// TIA Portal V20 export
FUNCTION_BLOCK "FB_LoaderFixture"   // FB207, SCL
{ S7_Optimized_Access := 'TRUE' }
// stored: AutoNumber false, MemoryReserve 100, SetENOAutomatically false
   VAR_INPUT
      iAxisV_Moving : Bool;
      iAxisV_InPos : Bool;
      iAxisW_Moving : Bool;
      iAxisW_InPos : Bool;
   END_VAR
   VAR_OUTPUT
      oFixtureOpenReq : Bool;
      oFixtureCloseReq : Bool;
      oLoadGripperOpenReq : Bool;
      oUnloadGripperCloseReq : Bool;
      oBlowingReq : Bool;
      oAxisV_StartReq : Bool;
      oAxisV_PosSetPoint : Real;
      oAxisW_StartReq : Bool;
      oAxisW_PosSetPoint : Real;
   END_VAR
   VAR
      sFixtureMain : "FB_FixtureUnloadLoad";
      sFixtureUnloading { S7_SetPoint := 'True'} : "FB_FixtureUnloading";
      sFixtureLoading { S7_SetPoint := 'True'} : "FB_FixtureLoading";
      sFixtureBlowing { S7_SetPoint := 'True'} : "FB_FixtureBlowing";
      sFixtureRelease { S7_SetPoint := 'True'} : "FB_FixtureRelease";
      sFixtureV_Init { S7_SetPoint := 'True'} : "FB_FixtureV_Init";
      sFixtureW_Init { S7_SetPoint := 'True'} : "FB_FixtureW_Init";
      sAxisVSafePos { S7_SetPoint := 'True'} : LReal;
      sStepPauseSeq { S7_SetPoint := 'True'} : Bool;
   END_VAR
   VAR_TEMP
      tAxisV_Position : Struct
         FixtureLoad : Bool;
         FixtureUnload : Bool;
         FixtureBlowing : Bool;
         FixtureSafe : Bool;
         ShuttleSafe : Bool;
         Shuttle1Blowing : Bool;
      END_STRUCT;
      tAxisW_Position : Struct
         FixtureLoad : Bool;
         FixtureUnload : Bool;
         FixtureBlowing : Bool;
         FixtureSafe : Bool;
         Approach : Bool;
      END_STRUCT;
   END_VAR
BEGIN
   REGION Axis V Safe Position
       IF "DB_LoaderShuttle1".sShuttlePosInt THEN
           #sAxisVSafePos := "DB_AxisPosMachinePLC".Axis_V.Shuttle_1.LoadUnload;
       ELSIF "DB_LoaderShuttle2".sShuttlePosInt THEN
           #sAxisVSafePos := "DB_AxisPosMachinePLC".Axis_V.Shuttle_2.LoadUnload;
       ELSE
           #sAxisVSafePos := "DB_AxisPosMachinePLC".Axis_V.Fixture.Safe;
       END_IF;
       // WFA revoir la gestion du Setpoint Safe en foncton de la shuttle
       #sAxisVSafePos := "DB_AxisPosMachinePLC".Axis_V.Fixture.Safe;
   END_REGION

   REGION Position Check
       REGION Axis V
           // Position : Fixture Load
           "FC_PositionCheck"(iAxisCurrentPos := "DB_AxisPosition".sAxis07_V."$AA_IM",
                              iAxisTargetPos := "DB_AxisPosMachinePLC".Axis_V.Fixture.Load,
                              iTolMin := 0.001,
                              iTolMax := 0.001,
                              iInPos => #tAxisV_Position.FixtureLoad);

           // Position : Fixture Unload
           "FC_PositionCheck"(iAxisCurrentPos := "DB_AxisPosition".sAxis07_V."$AA_IM",
                              iAxisTargetPos := "DB_AxisPosMachinePLC".Axis_V.Fixture.Unload,
                              iTolMin := 0.001,
                              iTolMax := 0.001,
                              iInPos => #tAxisV_Position.FixtureUnload);

           // Position : Fixture Blowing
           "FC_PositionCheck"(iAxisCurrentPos := "DB_AxisPosition".sAxis07_V."$AA_IM",
                              iAxisTargetPos := "DB_AxisPosMachinePLC".Axis_V.Fixture.Blowing,
                              iTolMin := 0.001,
                              iTolMax := 0.001,
                              iInPos => #tAxisV_Position.FixtureBlowing);

           // Position : Fixture Safe
           "FC_PositionCheck"(iAxisCurrentPos := "DB_AxisPosition".sAxis07_V."$AA_IM",
                              iAxisTargetPos := #sAxisVSafePos,
                              iTolMin := 0.001,
                              iTolMax := 0.001,
                              iInPos => #tAxisV_Position.FixtureSafe);

           // Position : Safe (Shuttle)
           "FC_PositionCheck"(iAxisCurrentPos := "DB_AxisPosition".sAxis07_V."$AA_IM",
                              iAxisTargetPos := "DB_AxisPosMachinePLC".Axis_V.Safe,
                              iTolMin := 0.001,
                              iTolMax := 0.001,
                              iInPos => #tAxisV_Position.ShuttleSafe);

           // Position : Blowing Shuttle 1
           "FC_PositionCheck"(iAxisCurrentPos := "DB_AxisPosition".sAxis07_V."$AA_IM",
                              iAxisTargetPos := "DB_AxisPosMachinePLC".Axis_V.Shuttle_1.Blowing,
                              iTolMin := 0.001,
                              iTolMax := 0.001,
                              iInPos => #tAxisV_Position.Shuttle1Blowing);
       END_REGION

       REGION Axis W
           // Position : Fixture Load
           "FC_PositionCheck"(iAxisCurrentPos := "DB_AxisPosition".sAxis08_W."$AA_IM",
                              iAxisTargetPos := "DB_AxisPosMachinePLC".Axis_W.Fixture.Load,
                              iTolMin := 0.001,
                              iTolMax := 0.001,
                              iInPos => #tAxisW_Position.FixtureLoad);

           // Position : Fixture Unload
           "FC_PositionCheck"(iAxisCurrentPos := "DB_AxisPosition".sAxis08_W."$AA_IM",
                              iAxisTargetPos := "DB_AxisPosMachinePLC".Axis_W.Fixture.Unload,
                              iTolMin := 0.001,
                              iTolMax := 0.001,
                              iInPos => #tAxisW_Position.FixtureUnload);

           // Position : Fixture Blowing
           "FC_PositionCheck"(iAxisCurrentPos := "DB_AxisPosition".sAxis08_W."$AA_IM",
                              iAxisTargetPos := "DB_AxisPosMachinePLC".Axis_W.Fixture.Blowing,
                              iTolMin := 0.001,
                              iTolMax := 0.001,
                              iInPos => #tAxisW_Position.FixtureBlowing);

           // Position : Fixture Safe
           "FC_PositionCheck"(iAxisCurrentPos := "DB_AxisPosition".sAxis08_W."$AA_IM",
                              iAxisTargetPos := "DB_AxisPosMachinePLC".Axis_W.Fixture.Safe,
                              iTolMin := 0.001,
                              iTolMax := 0.001,
                              iInPos => #tAxisW_Position.FixtureSafe);

           // Position : Approach (confondu avec load/unload)
           "FC_PositionCheck"(iAxisCurrentPos := "DB_AxisPosition".sAxis08_W."$AA_IM",
                              iAxisTargetPos := "DB_AxisPosMachinePLC".Axis_W.Fixture.Approach,
                              iTolMin := 0.001,
                              iTolMax := 0.001,
                              iInPos => #tAxisW_Position.Approach);
       END_REGION
   END_REGION

   REGION Step Pause Sequence
       #sStepPauseSeq := "LBP_ModeGroup".E_JOG OR "DB_ExtraMissingPart".sGlobalExtraMissing;

       #sFixtureUnloading.iStepPause := #sStepPauseSeq;
       #sFixtureLoading.iStepPause := #sStepPauseSeq;
       #sFixtureBlowing.iStepPause := #sStepPauseSeq;
       #sFixtureRelease.iStepPause := #sStepPauseSeq;
       #sFixtureV_Init.iStepPause := #sStepPauseSeq;
       #sFixtureW_Init.iStepPause := #sStepPauseSeq;
   END_REGION

   REGION Fixture Unload Load
       // M33 : Fixture Unloading Request
       #sFixtureMain.iFixtureUnloadingRequest := "LBP_Chan1".MDyn[33];

       // M35 : Fixture Blowing Request
       #sFixtureMain.iFixtureBlowingRequest := "LBP_Chan1".MDyn[35];

       // M34 : Fixture Loading Request
       #sFixtureMain.iFixtureLoadingRequest := "LBP_Chan1".MDyn[34];

       // Release request (Release not used)
       #sFixtureMain.iFixtureReleaseRequest := FALSE;

       // M31 : Fixture V Init Request
       #sFixtureMain.iFixtureV_InitRequest := "LBP_Chan1".MDyn[31];

       // M32 : Fixture W Init Request
       #sFixtureMain.iFixtureW_InitRequest := "LBP_Chan1".MDyn[32];

       // Gripper ready for unloading
       #sFixtureMain.iGripperReadyForUnloading := ("DB_GestionGripper".sGripperStatus.Available OR "DB_GestionGripper".sGripperStatus.DrivedByFixture)
       AND ((NOT "DB_PartManagement".sPosition.sGripper.Drilled.Presence.Part AND NOT "DB_PartManagement".sPosition.sGripper.Drilled.Presence.BW AND "DB_GestionGripper".sDrilledGripper.oStateOpen AND "DB_WorkingModes".sEmptying)
       OR (NOT "DB_PartManagement".sPosition.sGripper.Drilled.Presence.Part AND NOT "DB_PartManagement".sPosition.sGripper.Drilled.Presence.BW AND "DB_PartManagement".sPosition.sGripper.Undrilled.Presence.Part AND "DB_PartManagement".sPosition.sGripper.Undrilled.Presence.BW AND "DB_GestionGripper".sDrilledGripper.oStateOpen AND "DB_WorkingModes".sNormal));

       // Gripper ready for loading
       #sFixtureMain.iGripperReadyForLoading := ("DB_GestionGripper".sGripperStatus.Available OR "DB_GestionGripper".sGripperStatus.DrivedByFixture)
       AND (("DB_PartManagement".sPosition.sGripper.Undrilled.Presence.Part AND "DB_PartManagement".sPosition.sGripper.Undrilled.Presence.BW AND "DB_WorkingModes".sFilling)
       OR ("DB_PartManagement".sPosition.sGripper.Undrilled.Presence.Part AND "DB_PartManagement".sPosition.sGripper.Undrilled.Presence.BW  AND ("DB_WorkingModes".sNormal OR "DB_WorkingModes".sEmptying)));

       // Gripper ready for blowing
       #sFixtureMain.iGripperReadyForBlowing := ("DB_GestionGripper".sGripperStatus.Available OR "DB_GestionGripper".sGripperStatus.DrivedByFixture)
       AND #sFixtureMain.iGripperReadyForLoading;

       // Gripper ready for Release (Release not used)
       #sFixtureMain.iGripperReadyForRelease := ("DB_GestionGripper".sGripperStatus.Available OR "DB_GestionGripper".sGripperStatus.DrivedByFixture);

       // Gripper ready for V Init
       #sFixtureMain.iGripperReadyForV_Init := ("DB_GestionGripper".sGripperStatus.Available OR "DB_GestionGripper".sGripperStatus.DrivedByFixture);

       // Gripper ready for W Init
       #sFixtureMain.iGripperReadyForW_Init := ("DB_GestionGripper".sGripperStatus.Available OR "DB_GestionGripper".sGripperStatus.DrivedByFixture);


       // Fixture ready for unloading
       #sFixtureMain.iFixtureReadyForUnloading := TRUE;

       // Fixture ready for loading
       #sFixtureMain.iFixtureReadyForLoading := "DB_PartManagement".sPosition.sFixtureEmpty;

       // Fixture ready for blowing
       #sFixtureMain.iFixtureReadyForBlowing := TRUE;

       // Fixture ready for Release (Release not used)
       #sFixtureMain.iFixtureReadyForRelease := TRUE;

       // Fixture ready for V Init
       #sFixtureMain.iFixtureReadyForV_Init := TRUE;

       // Fixture ready for W Init
       #sFixtureMain.iFixtureReadyForW_Init := TRUE;


       // Axis ready for Unloading
       #sFixtureMain.iAxisReadyForUnloading :=
       ("DB_AxisPosition".sAxis01_X."$AA_IM" = "DB_AxisPosMachineNC".Axis_X.Unload
       AND "DB_AxisPosition".sAxis02_Y."$AA_IM" = "DB_AxisPosMachineNC".Axis_Y.Unload
       AND "DB_AxisPosition".sAxis04_B."$AA_IM" = "DB_AxisPosMachineNC".Axis_B.Unload
       AND "DB_AxisPosition".sAxis03_ZM."$AA_IM" = "DB_AxisPosition".sAxis03_ZM."$MA_POS_LIMIT_MINUS2" + 1);

       // Axis ready for Loading
       #sFixtureMain.iAxisReadyForLoading :=
       ("DB_AxisPosition".sAxis01_X."$AA_IM" = "DB_AxisPosMachineNC".Axis_X.Load
       AND "DB_AxisPosition".sAxis02_Y."$AA_IM" = "DB_AxisPosMachineNC".Axis_Y.Load
       AND "DB_AxisPosition".sAxis04_B."$AA_IM" = "DB_AxisPosMachineNC".Axis_B.Load
       AND "DB_AxisPosition".sAxis03_ZM."$AA_IM" = "DB_AxisPosition".sAxis03_ZM."$MA_POS_LIMIT_MINUS2" + 1);

       // Axis ready for Blowing
       #sFixtureMain.iAxisReadyForBlowing :=
       ("DB_AxisPosition".sAxis01_X."$AA_IM" = "DB_AxisPosMachineNC".Axis_X.Blowing
       AND "DB_AxisPosition".sAxis02_Y."$AA_IM" = "DB_AxisPosMachineNC".Axis_Y.Blowing
       AND "DB_AxisPosition".sAxis04_B."$AA_IM" = "DB_AxisPosMachineNC".Axis_B.Blowing
       AND "DB_AxisPosition".sAxis03_ZM."$AA_IM" = "DB_AxisPosition".sAxis03_ZM."$MA_POS_LIMIT_MINUS2" + 1);

       // Axis ready for Release (Release not used)
       #sFixtureMain.iAxisReadyForRelease :=
       ("DB_AxisPosition".sAxis03_ZM."$AA_IM" = "DB_AxisPosition".sAxis03_ZM."$MA_POS_LIMIT_MINUS2" + 1
       AND "DB_AxisPosition".sAxis09_ZL."$AA_IM" = "DB_AxisPosMachineNC".Axis_ZL.Safe);

       // Axis ready for V Init
       #sFixtureMain.iAxisReadyForV_Init := TRUE;

       // Axis ready for W Init
       #sFixtureMain.iAxisReadyForW_Init := TRUE;

       #sFixtureMain(iFixtureUnloadingRequest:=#sFixtureMain.iFixtureUnloadingRequest,
                     iFixtureLoadingRequest:=#sFixtureMain.iFixtureLoadingRequest,
                     iFixtureBlowingRequest:=#sFixtureMain.iFixtureBlowingRequest,
                     iFixtureReleaseRequest:=#sFixtureMain.iFixtureReleaseRequest,
                     iFixtureV_InitRequest:=#sFixtureMain.iFixtureV_InitRequest,
                     iFixtureW_InitRequest:=#sFixtureMain.iFixtureW_InitRequest,
                     iWorkingModeFilling:="DB_WorkingModes".sFilling,
                     iWorkingModeEmptying:="DB_WorkingModes".sEmptying,
                     iGripperReadyForUnloading:=#sFixtureMain.iGripperReadyForUnloading,
                     iGripperReadyForLoading:=#sFixtureMain.iGripperReadyForLoading,
                     iGripperReadyForBlowing:=#sFixtureMain.iGripperReadyForBlowing,
                     iGripperReadyForRelease:=#sFixtureMain.iGripperReadyForRelease,
                     iGripperReadyForV_Init:=#sFixtureMain.iGripperReadyForV_Init,
                     iGripperReadyForW_Init:=#sFixtureMain.iGripperReadyForW_Init,
                     iFixtureReadyForUnloading:=#sFixtureMain.iFixtureReadyForUnloading,
                     iFixtureReadyForLoading:=#sFixtureMain.iFixtureReadyForLoading,
                     iFixtureReadyForBlowing:=#sFixtureMain.iFixtureReadyForBlowing,
                     iFixtureReadyForRelease:=#sFixtureMain.iFixtureReadyForRelease,
                     iFixtureReadyForV_Init:=#sFixtureMain.iFixtureReadyForV_Init,
                     iFixtureReadyForW_Init:=#sFixtureMain.iFixtureReadyForW_Init,
                     iAxisReadyForUnloading:=#sFixtureMain.iAxisReadyForUnloading,
                     iAxisReadyForLoading:=#sFixtureMain.iAxisReadyForLoading,
                     iAxisReadyForBlowing:=#sFixtureMain.iAxisReadyForBlowing,
                     iAxisReadyForRelease:=#sFixtureMain.iAxisReadyForRelease,
                     iAxisReadyForV_Init:=#sFixtureMain.iAxisReadyForV_Init,
                     iAxisReadyForW_Init:=#sFixtureMain.iAxisReadyForW_Init,
                     iAxisV_W_Available:="DB_GestionGripper".sGripperStatus.Available,
                     oAxisV_W_Reservation=>"DB_GestionGripper".sGripperReq.ByFixture,
                     oNC_RID1=>"LBP_AlarmMsgs".Chan[1].RID[8],
                     oNC_RID2=>"LBP_AlarmMsgs".Chan[1].RID[9],
                     ioFixtureUnloadingSeq:=#sFixtureUnloading.sInterface,
                     ioFixtureLoadingSeq:=#sFixtureLoading.sInterface,
                     ioFixtureBlowingSeq:=#sFixtureBlowing.sInterface,
                     ioFixtureReleaseSeq:=#sFixtureRelease.sInterface,
                     ioFixtureV_InitSeq:=#sFixtureV_Init.sInterface,
                     ioFixtureW_InitSeq:=#sFixtureW_Init.sInterface);
   END_REGION

   REGION Fixture Unloading
       // Unload Gripper Closed according to dry run working mode
        #sFixtureUnloading.iUnloadGripperClosed := ("DB_GestionGripper".sDrilledGripper.oStateCloseWithPart AND NOT "DB_WorkingModes".sDryRun)
        OR ("DB_GestionGripper".sDrilledGripper.oStateClose AND "DB_WorkingModes".sDryRun);

       #sFixtureUnloading(iStartSeqCond:= "DB_PowerOn".sMachineReadySoft AND NOT "DB_LoaderFixtureMain".sUnloadingNotFinished AND NOT "MCP1_In".reset,
                          iJobReq:=#sFixtureUnloading.sInterface.StartRequest,
                          iFixtureOpened:="DB_DigitalInputs".sClampingOpenCtrl.sSWStatus,
                          iUnloadGripperClosed:=#sFixtureUnloading.iUnloadGripperClosed, // WAF CHECK
                          iAxisV_FixtUnloadPos:=#tAxisV_Position.FixtureUnload,
                          iAxisV_FixtUnloadPosSetPoint:="DB_AxisPosMachinePLC".Axis_V.Fixture.Unload,
                          iAxisW_FixtSafePos:=#tAxisW_Position.FixtureSafe,
                          iAxisW_FixtSafePosSetPoint:="DB_AxisPosMachinePLC".Axis_W.Fixture.Safe,
                          iAxisW_FixtUnloadPos:=#tAxisW_Position.FixtureUnload,
                          iAxisW_FixtUnloadPosSetPoint:="DB_AxisPosMachinePLC".Axis_W.Fixture.Unload,
                          iAxisV_Moving:=#iAxisV_Moving,
                          iAxisV_InPos:=#iAxisV_InPos,
                          iAxisW_Moving:=#iAxisW_Moving,
                          iAxisW_InPos:=#iAxisW_InPos,
                          iPLC_DateAndTime:="DB_ReadDateAndTime".sDateAndTime,
                          iStepPause:=#sFixtureUnloading.iStepPause,
                          oFixtureOpenReq=>#sFixtureUnloading.oFixtureOpenReq,
                          oUnloadGripperCloseReq=>#sFixtureUnloading.oUnloadGripperCloseReq,
                          oVacuumStopReq=>#sFixtureUnloading.oVacuumStopReq,
                          oAxisV_StartReq=>#sFixtureUnloading.oAxisV_StartReq,
                          oAxisV_PosSetPoint=>#sFixtureUnloading.oAxisV_PosSetPoint,
                          oAxisW_StartReq=>#sFixtureUnloading.oAxisW_StartReq,
                          oAxisW_PosSetPoint=>#sFixtureUnloading.oAxisW_PosSetPoint);
   END_REGION

   REGION Fixture Loading
       // Load Gripper Closed according to dry run working mode
       #sFixtureLoading.iFixtureClosed := ("DB_GestionFixture".sFixturePartControl.oGoodPart AND NOT "DB_WorkingModes".sDryRun)
       OR ("DB_DigitalOutputs".sClampingClosing.sSWStatus AND ("DB_WorkingModes".sDryRun));

       #sFixtureLoading(iStartSeqCond := "DB_PowerOn".sMachineReadySoft AND NOT "DB_LoaderFixtureMain".sLoadingNotFinished AND NOT "MCP1_In".reset,
                        iJobReq := #sFixtureLoading.sInterface.StartRequest,
                        iFixtureOpened := "DB_DigitalInputs".sClampingOpenCtrl.sSWStatus,
                        iFixtureClosed := #sFixtureLoading.iFixtureClosed,
                        iLoadGripperOpened := "DB_GestionGripper".sUndrilledGripper.oStateOpen,
                        iAxisV_FixtLoadPos := #tAxisV_Position.FixtureLoad,
                        iAxisV_FixtLoadPosSetPoint := "DB_AxisPosMachinePLC".Axis_V.Fixture.Load,
                        iAxisW_FixtSafePos := #tAxisW_Position.FixtureSafe,
                        iAxisW_FixtSafePosSetPoint := "DB_AxisPosMachinePLC".Axis_W.Fixture.Safe,
                        iAxisW_FixtLoadPos := #tAxisW_Position.FixtureLoad,
                        iAxisW_FixtLoadPosSetPoint := "DB_AxisPosMachinePLC".Axis_W.Fixture.Load,
                        iAxisW_FixtApproachPos:=#tAxisW_Position.Approach,
                        iAxisW_FixtApproachPosSetPoint:="DB_AxisPosMachinePLC".Axis_W.Fixture.Approach,
                        iAxisV_Moving := #iAxisV_Moving,
                        iAxisV_InPos := #iAxisV_InPos,
                        iAxisW_Moving := #iAxisW_Moving,
                        iAxisW_InPos := #iAxisW_InPos,
                        iPLC_DateAndTime := "DB_ReadDateAndTime".sDateAndTime,
                        iStepPause := #sFixtureLoading.iStepPause,
                        oFixtureOpenReq => #sFixtureLoading.oFixtureOpenReq,
                        oFixtureCloseReq => #sFixtureLoading.oFixtureCloseReq,
                        oLoadGripperOpenReq => #sFixtureLoading.oLoadGripperOpenReq,
                        oVacuumStartReq=>#sFixtureLoading.oVacuumStartReq,
                        oAxisV_StartReq => #sFixtureLoading.oAxisV_StartReq,
                        oAxisV_PosSetPoint => #sFixtureLoading.oAxisV_PosSetPoint,
                        oAxisW_StartReq => #sFixtureLoading.oAxisW_StartReq,
                        oAxisW_PosSetPoint => #sFixtureLoading.oAxisW_PosSetPoint);
   END_REGION

   REGION Fixture Blowing
       #sFixtureBlowing(iStartSeqCond:= "DB_PowerOn".sMachineReadySoft AND NOT "DB_LoaderFixtureMain".sBlowingNotFinished AND NOT "MCP1_In".reset,
                        iJobReq:=#sFixtureBlowing.sInterface.StartRequest,
                        iFixtureOpened:="DB_DigitalInputs".sClampingOpenCtrl.sSWStatus,
                        iAxisV_FixtBlowingPos:=#tAxisV_Position.FixtureBlowing,
                        iAxisV_FixtBlowingPosSetPoint:="DB_AxisPosMachinePLC".Axis_V.Fixture.Blowing,
                        iAxisW_FixtSafePos:=#tAxisW_Position.FixtureSafe,
                        iAxisW_FixtSafePosSetPoint:="DB_AxisPosMachinePLC".Axis_W.Fixture.Safe,
                        iAxisW_FixtBlowPos:=#tAxisW_Position.FixtureBlowing,
                        iAxisW_FixtBlowPosSetPoint:="DB_AxisPosMachinePLC".Axis_W.Fixture.Blowing,
                        iAxisV_Moving:=#iAxisV_Moving,
                        iAxisV_InPos:=#iAxisV_InPos,
                        iAxisW_Moving:=#iAxisW_Moving,
                        iAxisW_InPos:=#iAxisW_InPos,
                        iBlowingTime:= DINT_TO_TIME(REAL_TO_DINT("DB_HMISetting".BlowingSetpoint)),
                        iPLC_DateAndTime:="DB_ReadDateAndTime".sDateAndTime,
                        iStepPause:=#sFixtureBlowing.iStepPause,
                        oFixtureOpenReq=>#sFixtureBlowing.oFixtureOpenReq,
                        oAxisV_StartReq=>#sFixtureBlowing.oAxisV_StartReq,
                        oAxisV_PosSetPoint=>#sFixtureBlowing.oAxisV_PosSetPoint,
                        oAxisW_StartReq=>#sFixtureBlowing.oAxisW_StartReq,
                        oAxisW_PosSetPoint=>#sFixtureBlowing.oAxisW_PosSetPoint,
                        oBlowingReq=>#sFixtureBlowing.oBlowingReq);
   END_REGION

   REGION Fixture Release  (Release not used)
       // Repli en position
       //  - Shuttle 1 (Pos. blowing Shuttle 1)
       //  - Shuttle 2 ( Pos Safe)
       IF "DB_LoaderShuttle1".sMain.sCurrent_Step_NB = 70 THEN
           #sFixtureRelease.iAxisV_SafePos := #tAxisV_Position.Shuttle1Blowing;
           #sFixtureRelease.iAxisV_SafePosSetPoint := "DB_AxisPosMachinePLC".Axis_V.Shuttle_1.Blowing;
       ELSE
           #sFixtureRelease.iAxisV_SafePos := #tAxisV_Position.ShuttleSafe;
           #sFixtureRelease.iAxisV_SafePosSetPoint := "DB_AxisPosMachinePLC".Axis_V.Safe;
       END_IF;

       #sFixtureRelease(iStartSeqCond := "DB_PowerOn".sMachineReadySoft AND NOT "DB_LoaderFixtureMain".sReleaseNotFinished AND NOT "MCP1_In".reset, // WAF TBD
                        iJobReq := #sFixtureRelease.sInterface.StartRequest,
                        iAxisV_SafePos := #sFixtureRelease.iAxisV_SafePos, // #tAxis_V_Position.Shuttle1Blowing, // #tAxis_V_Position.ShuttleSafe,
                        iAxisV_SafePosSetPoint := #sFixtureRelease.iAxisV_SafePosSetPoint, // "DB_AxisPosMachinePLC".Axis_V.Shuttle_1.Blowing,     // "DB_AxisPosMachinePLC".Axis_V.Safe,
                        iAxisW_FixtSafePos := #tAxisW_Position.FixtureSafe,
                        iAxisW_FixtSafePosSetPoint := "DB_AxisPosMachinePLC".Axis_W.Fixture.Safe,
                        iAxisV_Moving := #iAxisV_Moving,
                        iAxisV_InPos := #iAxisV_InPos,
                        iAxisW_Moving := #iAxisW_Moving,
                        iAxisW_InPos := #iAxisW_InPos,
                        iPLC_DateAndTime := "DB_ReadDateAndTime".sDateAndTime,
                        iStepPause := #sFixtureRelease.iStepPause,
                        oAxisV_StartReq => #sFixtureRelease.oAxisV_StartReq,
                        oAxisV_PosSetPoint => #sFixtureRelease.oAxisV_PosSetPoint,
                        oAxisW_StartReq => #sFixtureRelease.oAxisW_StartReq,
                        oAxisW_PosSetPoint => #sFixtureRelease.oAxisW_PosSetPoint);
   END_REGION

   REGION Fixture V Init
       #sFixtureV_Init(iStartSeqCond := "DB_PowerOn".sMachineReadySoft AND NOT "DB_LoaderFixtureMain".sV_InitNotFinished AND NOT "MCP1_In".reset,
                       iJobReq := #sFixtureV_Init.sInterface.StartRequest,
                       iAxisV_FixtSafePos := #tAxisV_Position.FixtureSafe,
                       iAxisV_FixtSafePosSetPoint := #sAxisVSafePos,
                       iAxisV_Moving := #iAxisV_Moving,
                       iAxisV_InPos := #iAxisV_InPos,
                       iPLC_DateAndTime := "DB_ReadDateAndTime".sDateAndTime,
                       iStepPause := #sFixtureV_Init.iStepPause,
                       oAxisV_StartReq => #sFixtureV_Init.oAxisV_StartReq,
                       oAxisV_PosSetPoint => #sFixtureV_Init.oAxisV_PosSetPoint);
   END_REGION

   REGION Fixture W Init
       #sFixtureW_Init(iStartSeqCond := "DB_PowerOn".sMachineReadySoft AND NOT "DB_LoaderFixtureMain".sW_InitNotFinished AND NOT "MCP1_In".reset,
                       iJobReq := #sFixtureW_Init.sInterface.StartRequest,
                       iAxisW_FixtSafePos := #tAxisW_Position.FixtureSafe,
                       iAxisW_FixtSafePosSetPoint := "DB_AxisPosMachinePLC".Axis_W.Fixture.Safe,
                       iAxisW_Moving := #iAxisW_Moving,
                       iAxisW_InPos := #iAxisW_InPos,
                       iPLC_DateAndTime := "DB_ReadDateAndTime".sDateAndTime,
                       iStepPause := #sFixtureW_Init.iStepPause,
                       iAxisW_StartReq => #sFixtureW_Init.iAxisW_StartReq,
                       iAxisW_PosSetPoint => #sFixtureW_Init.iAxisW_PosSetPoint);
   END_REGION

   REGION Axis U-V-W Start Request  
       // Axis V - Start Request
       #oAxisV_StartReq :=
       #sFixtureUnloading.oAxisV_StartReq
       OR #sFixtureLoading.oAxisV_StartReq
       OR #sFixtureBlowing.oAxisV_StartReq
       OR #sFixtureRelease.oAxisV_StartReq
       OR #sFixtureV_Init.oAxisV_StartReq;

       // Axis V - Position Set point  according to start request
       IF #sFixtureUnloading.oAxisV_StartReq THEN
           #oAxisV_PosSetPoint := #sFixtureUnloading.oAxisV_PosSetPoint;
       ELSIF #sFixtureLoading.oAxisV_StartReq THEN
           #oAxisV_PosSetPoint := #sFixtureLoading.oAxisV_PosSetPoint;
       ELSIF #sFixtureBlowing.oAxisV_StartReq THEN
           #oAxisV_PosSetPoint := #sFixtureBlowing.oAxisV_PosSetPoint;
       ELSIF #sFixtureRelease.oAxisV_StartReq THEN
           #oAxisV_PosSetPoint := #sFixtureRelease.oAxisV_PosSetPoint;
       ELSIF #sFixtureV_Init.oAxisV_StartReq THEN
           #oAxisV_PosSetPoint := #sFixtureV_Init.oAxisV_PosSetPoint;
       ELSE
           #oAxisV_StartReq := FALSE;
       END_IF;

       // Axis W - Start Request
       #oAxisW_StartReq :=
       #sFixtureUnloading.oAxisW_StartReq
       OR #sFixtureLoading.oAxisW_StartReq
       OR #sFixtureBlowing.oAxisW_StartReq
       OR #sFixtureRelease.oAxisW_StartReq
       OR #sFixtureW_Init.iAxisW_StartReq;

       // Axis W - Position Set point  according to start request
       IF #sFixtureUnloading.oAxisW_StartReq THEN
           #oAxisW_PosSetPoint := #sFixtureUnloading.oAxisW_PosSetPoint;
       ELSIF #sFixtureLoading.oAxisW_StartReq THEN
           #oAxisW_PosSetPoint := #sFixtureLoading.oAxisW_PosSetPoint;
       ELSIF #sFixtureBlowing.oAxisW_StartReq THEN
           #oAxisW_PosSetPoint := #sFixtureBlowing.oAxisW_PosSetPoint;
       ELSIF #sFixtureRelease.oAxisW_StartReq THEN
           #oAxisW_PosSetPoint := #sFixtureRelease.oAxisW_PosSetPoint;
       ELSIF #sFixtureW_Init.iAxisW_StartReq THEN
           #oAxisW_PosSetPoint := #sFixtureW_Init.iAxisW_PosSetPoint;
       ELSE
           #oAxisW_StartReq := FALSE;
       END_IF;
   END_REGION


   REGION Gripper Command Request
       // Load Gripper
       #oLoadGripperOpenReq := #sFixtureLoading.oLoadGripperOpenReq;
       // Unload Gripper
       #oUnloadGripperCloseReq := #sFixtureUnloading.oUnloadGripperCloseReq;
   END_REGION

   REGION Fixture Command Request
       #oFixtureOpenReq := #sFixtureUnloading.oFixtureOpenReq
       OR #sFixtureLoading.oFixtureOpenReq
       OR #sFixtureBlowing.oFixtureOpenReq;

       #oFixtureCloseReq := #sFixtureLoading.oFixtureCloseReq;
   END_REGION

   REGION Blowing Command Request
       #oBlowingReq := #sFixtureBlowing.oBlowingReq;
   END_REGION

   REGION Message Waiting for Product
       "LBP_AlarmMsgs".UserA[03].A70UUxx[48] := #sFixtureMain.oNC_RID1;
   END_REGION
END_FUNCTION_BLOCK
